(* IEC 61131-3 sources: AXOpen/src/components.rexroth.drives/ctrl/src/AxoIndraDrive/TypesStructuresAndEnums, 10 files *)

(* ---- AxoIndraDriveErrorStruct.st ---- *)
NAMESPACE AXOpen.Components.Rexroth.Drives
    TYPE
        {S7.extern=ReadWrite}
        AxoIndraDriveErrorStruct :
        STRUCT
            Table       : AXOpen.Components.Rexroth.Drives.eAxoIndraDriveErrorTable;          (* Additional diagnosis table           *)
            Additional1 : DWORD;                (* Additional diagnosis number1         *)
            Additional2 : DWORD;                (* Additional diagnosis number2         *)
        END_STRUCT;
    END_TYPE
END_NAMESPACE

(* ---- eAxoIndraDriveErrorCode.st ---- *)
NAMESPACE AXOpen.Components.Rexroth.Drives
    TYPE PUBLIC
        eAxoIndraDriveErrorCode : WORD
        (
            NONE_ERROR                  := WORD#16#0000,     (* No error code available              *)
            (*                  invalid input                                                   *)
            INPUT_INVALID_ERROR         := WORD#16#0001,     (* Invalid input                        *)
            (*                  communications error                                            *)
            COMMUNICATION_ERROR         := WORD#16#0002,     (* Error while communication            *)
            (*                  data processing error                                           *)
            RESOURCE_ERROR              := WORD#16#0003,     (* Resource error                       *)
            ACCESS_ERROR                := WORD#16#0004,     (* Access error                         *)
            STATE_MACHINE_ERROR         := WORD#16#0005,     (* Invalid state State - Machine        *)
            INPUT_RANGE_ERROR           := WORD#16#0006,     (* Error because Input out of range     *)
            CALCULATION_ERROR           := WORD#16#0007,     (* Error while calculation              *)
            (*                  device error                                                    *)
            DEVICE_ERROR                := WORD#16#0008,     (* Device Error occurred                *)
            (*                  other error                                                     *)
            OTHER_ERROR                 := WORD#16#7FFE,     (* Undefined Error                      *)
            (*                  system error                                                    *)
            SYSTEM_ERROR                := WORD#16#7FFF      (* System error occured                 *)

                );
    END_TYPE
END_NAMESPACE

(* ---- eAxoIndraDriveErrorTable.st ---- *)
NAMESPACE AXOpen.Components.Rexroth.Drives
    TYPE PUBLIC
        eAxoIndraDriveErrorTable : WORD
        (
            NO_TABLE_USED           := WORD#16#0000,         //reserved
            SERCOS_TABLE            := WORD#16#0010,         //Sercos Error: Addtitional1 = Sercos Code
            MLDS_TABLE              := WORD#16#0020,         //Drive-based Motion - Logic
            MLC_TABLE               := WORD#16#0030,         //Controller - based Motion - Logic
            MTX_TABLE               := WORD#16#0040,         //CNC
            MLP_TABLE               := WORD#16#0050,         //PC  - based Motion Logic
            PLC_TABLE               := WORD#16#0060,         //PLC
            INDRV_TABLE             := WORD#16#0070,         //IndraDrive
            DIAX_TABLE              := WORD#16#0080,         //DIAX
            ECO_TABLE               := WORD#16#0090,         //EcoDrive
            PB_DP_TABLE             := WORD#16#0130,         //Profibus
            DEVICENET_TABLE         := WORD#16#0140,         //DeviceNet
            ETHERNET_TABLE          := WORD#16#0150,         //Ethernet
            INTERBUS_TABLE          := WORD#16#0160,         //Interbus
            F_RELATED_TABLE         := WORD#16#0170,         //function related
            USER1_TABLE             := WORD#16#1000,         //free User Table
            USER2_TABLE             := WORD#16#1001,         //free User Table
            USER3_TABLE             := WORD#16#1002,         //free User Table
            USER4_TABLE             := WORD#16#1003,         //free User Table
            USER5_TABLE             := WORD#16#1004,         //free User Table
            USER6_TABLE             := WORD#16#1005,         //free User Table
            USER7_TABLE             := WORD#16#1006,         //free User Table
            USER8_TABLE             := WORD#16#1007,         //free User Table
            USER9_TABLE             := WORD#16#1008,         //free User Table
            USER10_TABLE            := WORD#16#1009          //free User Table
        );
    END_TYPE
END_NAMESPACE

(* ---- AxoIndraDrive_Component_Status.st ---- *)
NAMESPACE AXOpen.Components.Rexroth.Drives
    {S7.extern=ReadWrite}
    {#ix-attr:[Container(Layout.Stack)]}
    // CLASS PUBLIC AxoIndraDrive_Component_Status EXTENDS AXOpen.Components.Abstractions.AxoComponent_Status
    //     VAR PUBLIC

    //     END_VAR
    // END_CLASS
    CLASS PUBLIC AxoIndraDrive_Component_Status EXTENDS AXOpen.Components.Drives.AxoDrive_Status
        VAR PUBLIC

        END_VAR
    END_CLASS
END_NAMESPACE

(* ---- AxoIndraDriveAxisData.st ---- *)
NAMESPACE AXOpen.Components.Rexroth.Drives
    {S7.extern=ReadWrite}
    CLASS AxoIndraDriveAxisData
        VAR PUBLIC
            (* Commands *)
            CallAxis					:	BOOL;			//Call axis method for cyclic communication
            ReadOnlyData				:	BOOL;			//Read only data values from drive
            CallNumberCyclic			:	INT :=-1; 		//Number of method call's for cyclic communication
            WriteCommand				:	BOOL;			//Write command to drive
            PowerOnReq					:	BOOL;			//Request to power the drive on
            ResetReq					:	BOOL;			//Request to reset the drive
            HomingReq					:	BOOL;			//Request to start homing
            JogPositiveReq				:	BOOL;			//Request to jog the drive in positive direction
            JogNegativeReq				:	BOOL;			//Request to jog the drive in negative direction
            DriveStopReq				:	BOOL;			//Set Drive Stop with writing deceleration value to drive
            DriveHaltReq				:	BOOL;			//Set Drive Halt with writing deceleration value to drive
            MoveVelocityReq				:	BOOL;			//Command is velocity
            TorqueControlReq			:	BOOL;			//Command is torque
            Relative					:	BOOL; 			//Move relative to (last recommended) positioning command value
            Additive					:	BOOL; 			//Move additive to actual position; works only if relative possitioning active
            Position					:	LREAL;			//Target position for the motion  (negative or positive)
            Velocity					:	LREAL;			//Value of the maximum velocity (always positive) (not necessarily reached) [u/s].
            Acceleration				:	LREAL;			//Value of the acceleration (always positive) (increasing energy of the motor) [u/s2]
            Deceleration				:	LREAL;			//Value of the deceleration (always positive) (decreasing energy of the motor) [u/s2]
            Jerk						:	LREAL;			//Value of the jerk (always positive) [u/s3]
            Torque						:	LREAL;			//Value of the torque (always positive)
            S_0_0144_SignalStateWord	: 	WORD;			//S-0-0144 SignalStateWord*)
            CallAxisParameterMethod		:	BOOL;			//Call axis method for parameter read/write
            EnableAcyclicCommunication	:	BOOL;			//Enable acyclic communication (for parameter read/write)
            CallNumberAcyclic			:	INT;			//Number of method call's for acyclic communication
            WriteParameter				:	BOOL;			//FALSE = read, TRUE  = write Value of selected Parameter
            SelectDataType				:	UINT;			//0= Bool, 1 = Any, 2 = REAL
            ParameterNumber				:	DINT;			//Parameter number
            WriteValueLint				:	LINT;			//DINT value to be written
            WriteValueReal				:	REAL;			//REAL value to be written
            OverrideVelocityFactor		:	LREAL := 1.0;	//LREAL value to be written
            OverrideAccelerationFactor	:	LREAL := 1.0;	//LREAL value to be written
            OverrideJerkFactor			:	LREAL := 1.0;	//LREAL value to be written
        (* States *)
            CommandWriteActive			:	BOOL; 			//Command transfer to drive is active
            SetpointReached				: 	BOOL;			//Setpoint reached
            PowerOK						:	BOOL; 			//Power OK
            HomeOK						:	BOOL;			//Drive has reached the homeposition
            ResetOK						:	BOOL; 			//Reset done
            HomingRunning				:	BOOL;			//Homing is active
            Stopped						:	BOOL; 			//Drive in stopped regularly
            Standstill					:	BOOL; 			//Drive in standstill
            InPosition					:	BOOL; 			//Drive in position
            StoppedDueError				:	BOOL; 			//Drive in stop due to error
            MessageActive				:	BOOL;			//Class 3 diagnostics (message) present
            WarningActive				:	BOOL;			//Class 2 diagnostics (warning) present
            FailureActive				:	BOOL;			//Class 1 diagnostics (failure) present
            PowerError					:	BOOL; 			//Power-Failure
            StopError					:	BOOL;			//Stopping-Failure
            ContinuousMotion			:	BOOL; 			//Continius motion
            DiscreteMotion				:	BOOL; 			//Discrete motion
            SynchronizedMotion			:	BOOL;			//Synchronized motion
            Error						:	BOOL;			//Error
            ErrorID						:	AXOpen.Components.Rexroth.Drives.eAxoIndraDriveErrorCode;		//Error identification, ErrorCode
            ErrorIdent					:	AXOpen.Components.Rexroth.Drives.AxoIndraDriveErrorStruct;	//Error identification
            ActualPosition				:	LREAL; 			//Shows actual position
            ActualVelocity				:	LREAL; 			//Shows actual velocity
            ActualTorque				:	LREAL; 			//Shows actual torque
            CheckAccessOK				:	BOOL := TRUE;	//Flag for checking valid access at Axis_Data array
            S_0_0145_SignalControlWord	:	WORD;			//S-0-0145 wSignalControlWord, **** exept bit 0 *****)

            DoneAcyclicCommunication 	:	BOOL; 			//Reading/writing of the individual parameter completed, output variables valid
            ActiveAcyclicCommunication	: 	BOOL; 			//Reading/writing of the individual parameter active, output variables invalid
            DecimalPlaces 				:	UINT;			//Decimal places of the selected parameters
            DataTypeRead				:	UINT; 			//Read data type of the selected parameters
            DataLengthRead				:	UINT;			//Length of the read parameters
            ReadValueDint				:	DINT;			//DINT Operating value of the individual parameter without weighting
            ReadValueReal				:	REAL;			//REAL weighted operating value
            Error_AcyclicCommunication	:	BOOL := FALSE;  //Error
            ErrorID_AcyclicCommunication:   AXOpen.Components.Rexroth.Drives.eAxoIndraDriveErrorCode;		//Error identification, ErrorCode
            ErrorIdent_AcyclicCommunication:AXOpen.Components.Rexroth.Drives.AxoIndraDriveErrorStruct; 	//Error identification
            hwIdDevice                  :   UINT;
            hwIdParamCh_IDN             :   UINT;
            hwID_F_ModulNotUsed         :   UINT;
            hwIdInput_9_Words           :   UINT;
            hwIdOutput_13_Words         :   UINT;

        END_VAR

    END_CLASS

END_NAMESPACE

(* ---- AxoIndraDriveAxisReference.st ---- *)
// USING AXOpen.Components.Drives;

NAMESPACE AXOpen.Components.Rexroth.Drives
    {S7.extern=ReadWrite}
    CLASS AxoIndraDriveAxisReference IMPLEMENTS AXOpen.Components.Abstractions.Drives.IAxoAxisReference
        VAR PUBLIC
            FieldBus_In     :   AXOpen.Components.Rexroth.Drives.AxoIndraDriveFieldBusIn;
            FieldBus_Out    :   AXOpen.Components.Rexroth.Drives.AxoIndraDriveFieldBusOut;
            Parameter_In    :   AXOpen.Components.Rexroth.Drives.AxoIndraDriveParameterIn;
            Parameter_Out   :   AXOpen.Components.Rexroth.Drives.AxoIndraDriveParameterOut;
            Data            :   AXOpen.Components.Rexroth.Drives.AxoIndraDriveAxisData;
            Config          :   AXOpen.Components.Drives.AxoDrive_Config;
            Status          :   AXOpen.Components.Drives.AxoDrive_Status;
        END_VAR
    END_CLASS
END_NAMESPACE

(* ---- AxoIndraDriveFieldBusIn.st ---- *)
NAMESPACE AXOpen.Components.Rexroth.Drives
    {S7.extern=ReadWrite}
    CLASS AxoIndraDriveFieldBusIn
        (******************* Drive configuration  ***********************
        Master communication; Fieldbus settings:

                Profile type: * free configurable mode*
                    Configuration of realtime channel:
                        realtime input (configured feedback values):	    (9words)
                                P-0-4078 Fieldbus status WORD               (2bytes)
                                S-0-0051 Position feedback 1 value          (4bytes)
                                S-0-0040 Veloccity feedback value           (4bytes)
                                S-0-0390 Diagnostig message number          (4bytes)
                                S-0-0144 Signal status  word			    (2bytes)
                                S-0-0084 Actual torque/force value          (2bytes)
                        realtime output (configured command values):		(13words)
                                P-0-4077 Fieldbus control WORD              (2bytes)
                                S-0-0282 Positioning command value          (4bytes)
                                S-0-0259 Positioning velocity value         (4bytes)
                                S-0-0260 Positioning Accelelration          (4bytes)
                                S-0-0359 Positioning Deceleration           (4bytes)
                                S-0-0145 Signal control word                (2bytes)
                                S-0-0080 Torque/force command value		    (2bytes)
                                S-0-0193 Positioning jerk                   (4bytes)
                General settings:
                        S-0-0027, Configuration list signal control word -> Number 0; Content S-0-0393
                        S-0-0329, Assign list signal control word -> Number 0; Content 2
                        Primary operation mode: Drive controlled positioning, encoder 1 (without axis control word)
                        Secondary operation mode: Torque/force control
        *)
        VAR PUBLIC
            PhaseAcknowledgeBit0		:	BOOL;		//Operating mode acknowledge bit 0
            PhaseAcknowledgeBit1 		:	BOOL;		//Operating mode acknowledge bit 1
            InReference 				:	BOOL;		//In reference
            InStandstill 				:	BOOL;		//In standstill
            SetpointReached				:	BOOL;		//Setpoint reached
            CommandChangeBit 			:	BOOL;		//Command change bit
            OperatingModeError 			:	BOOL;		//Operating mode_error
            StatusSetpointProcess 		:	BOOL;		//Status setpoint processing
            ActualOperatingModeBit0 	:	BOOL;		//Actual_operating mode bit 0
            ActualOperatingModeBit1 	:	BOOL;		//Actual_operating mode bit 1
            SetpointAcknowledge 		:	BOOL;		//Setpoint acknowledge
            MessageZKL3 				:	BOOL;		//Message ZKL3
            WarningZKL2 				:	BOOL;		//Warning ZKL2
            DriveErrorZKL1 				:	BOOL;		//Drive Error ZKL1
            ReadyToOperateBit0 			:	BOOL;		//Ready to operate bit 0
            ReadyToOperateBit1 			:	BOOL;		//Ready to operate bit 1
            S_0_0051_ActualPosition		:	DWORD;		//Actual position
            S_0_0040_ActualVelocity		:	DWORD;		//Actual velocity
            S_0_0390_Diagnosis			:	DWORD;		//Diagnosis
            S_0_0144_SignalStatusWord	:	WORD;		//Signal status word
            S_0_0084_ActualTorque 		:	WORD;		//Actual torque
        END_VAR
    END_CLASS

END_NAMESPACE

(* ---- AxoIndraDriveFieldBusOut.st ---- *)
NAMESPACE AXOpen.Components.Rexroth.Drives
    {S7.extern=ReadWrite}
    CLASS AxoIndraDriveFieldBusOut
        (******************* Drive configuration  ***********************
        Master communication; Fieldbus settings:

                Profile type: * free configurable mode*
                    Configuration of realtime channel:
                        realtime input (configured feedback values):	    (9words)
                                P-0-4078 Fieldbus status WORD               (2bytes)
                                S-0-0051 Position feedback 1 value          (4bytes)
                                S-0-0040 Veloccity feedback value           (4bytes)
                                S-0-0390 Diagnostig message number          (4bytes)
                                S-0-0144 Signal status  word			    (2bytes)
                                S-0-0084 Actual torque/force value          (2bytes)
                        realtime output (configured command values):		(13words)
                                P-0-4077 Fieldbus control WORD              (2bytes)
                                S-0-0282 Positioning command value          (4bytes)
                                S-0-0259 Positioning velocity value         (4bytes)
                                S-0-0260 Positioning Accelelration          (4bytes)
                                S-0-0359 Positioning Deceleration           (4bytes)
                                S-0-0145 Signal control word                (2bytes)
                                S-0-0080 Torque/force command value		    (2bytes)
                                S-0-0193 Positioning jerk                   (4bytes)
                General settings:
                        S-0-0027, Configuration list signal control word -> Number 0; Content S-0-0393
                        S-0-0329, Assign list signal control word -> Number 0; Content 2
                        Primary operation mode: Drive controlled positioning, encoder 1 (without axis control word)
                        Secondary operation mode: Torque/force control
        *)
        VAR PUBLIC
            SetpointAcceptance 				:	BOOL;			//Setpoint acceptance
            OperatingModeSet 				:	BOOL;			//Operating mode set
            DriveToZeroPoint 				:	BOOL;			//Drive to zero point
            AbsoluteRelative 				:	BOOL;			//Position absolute = 0 or relative = 1
            ImmediateBlockChange 			:	BOOL;			//Immediate change
            ErrorDelete 					:	BOOL;			//Clear error
            JogForward 						:	BOOL;			//Jog forward
            JogBackward 					:	BOOL;			//Jog backward
            SetOperatingModeBit0 			:	BOOL;			//Setpoint operating mode_bit0
            SetOperatingModeBit1 			:	BOOL;			//Setpoint operating mode_bit1
            Iposync 						:	BOOL;			//Only in cycl. pos. control
            DriveHalt 						:	BOOL;			//Drive halt
            DriveEnable 					:	BOOL;			//Drive enable
            DriveOn 						:	BOOL;			//Drive on
            S_0_0282_CommandPosition		: 	DWORD;			//Command position
            S_0_0259_CommandVelocity		: 	DWORD;          //Command velocity
            S_0_0260_CommandAcceleration	: 	DWORD;          //Command acceleration
            S_0_0359_CommandDecceleration	: 	DWORD;          //Command decceleration
            S_0_0145_SignalControlWord		: 	WORD;           //Signal control word
            S_0_0080_TorqueForceCommand     :   WORD;           //Torque/force command value
            S_0_0193_CommandJerk            :   DWORD;          //Command jerk
        END_VAR
    END_CLASS
END_NAMESPACE

(* ---- AxoIndraDriveParameterIn.st ---- *)
NAMESPACE AXOpen.Components.Rexroth.Drives
    {S7.extern=ReadWrite}
    CLASS AxoIndraDriveParameterIn
        (******************* IndraDrive configuration  ***********************
        Master communication; Fieldbus settings:
        Parameter chanel 10Bytes / 5 Words I/O
        *)
        VAR PUBLIC
            Datalength	:	BYTE;	//Length of  transfer data*)
            FL_0		:	BOOL;	//Length userdata bit 0
            FL_1		:	BOOL;	//Length userdata bit 1
            FL_2		:	BOOL;	//Length userdata bit 2
            FL_3		:	BOOL;	//Length userdata bit 3
            ToggleBit	:	BOOL;	//Toggle bit
            LastBit		:	BOOL;	//Last bit
            Failure		:	BOOL;	//Failure while communication
            Reserve		:	BOOL;	//Reserve
            DataWord_0	:	WORD;	//Data WORD 0
            DataWord_1	:	WORD;	//Data word 1
            DataWord_2	:	WORD;	//Data word 2
            DataWord_3	:	WORD;	//Data word 3
        END_VAR
    END_CLASS
 END_NAMESPACE

(* ---- AxoIndraDriveParameterOut.st ---- *)
NAMESPACE AXOpen.Components.Rexroth.Drives
    {S7.extern=ReadWrite}
    CLASS AxoIndraDriveParameterOut
        (******************* IndraDrive configuration  ***********************
        Master communication; Fieldbus settings:
        Parameter chanel 10Bytes / 5 Words I/O
        *)
        VAR PUBLIC
            Datalength		:	BYTE := BYTE#04;//Length of transfer data
            FL_0			:	BOOL;			//Length userdata bit 0
            FL_1			:	BOOL;			//Length userdata bit 1
            FL_2			:	BOOL;			//Length userdata bit 2
            FL_3			:	BOOL;			//Length userdata bit 3
            ToggleBit		:	BOOL;			//Toggle bit
            LastBit			:	BOOL;			//Last bit
            Initalisation	:	BOOL := TRUE;	//Initialisation
            Reserve			:	BOOL;			//Reserve
            Index			:	WORD;			//Index number
            Subindex		:	BYTE;			//Subindex number
            Axis			:	BYTE;			//Axis number
            DataWord_0		:	WORD;			//Data word 0
            DataWord_1		:	WORD;			//Data word 1
        END_VAR
    END_CLASS
END_NAMESPACE
